// TIA Portal V19 export
FUNCTION "TolWin_REAL" : Bool   // FC70, LAD
// stored: Access Published, SetENOAutomatically false
   VAR_INPUT
      ActPos : Real;
      Target : Real;
      PosWin : Real;
   END_VAR
BEGIN

REGION Network 2 (SCL)
   #TolWin_REAL := ABS_LREAL(#ActPos - #Target) <= #PosWin;
END_REGION
END_FUNCTION
